(* IEC 61131-3 sources: beckhoffAutomationInterface/ST/Shark/Lib/Controllers/Temperature, 7 files *)

(* ---- GVL_HeatZone.st ---- *)
(* Compile-time bounds for FB_HeatZone arrays.
   MAX_CHANNELS sizes the per-zone channel arrays (the zone's _aipChannels).
   A "channel" is one RTD + one SSR + one PID controller pair.
   Pick the smallest bound that covers the largest physical heat zone on any
   supported machine. PRO DALP currently has 7 channels; 8 leaves headroom. *)
{attribute 'qualified_only'}
VAR_GLOBAL CONSTANT
    MAX_CHANNELS : INT := 8;   // Maximum channels per heat zone
END_VAR

(* ---- FB_BeckhoffTempController.st ---- *)
(* Beckhoff temperature controller for single heating zone. Integrates dual sensor support, PID control, and safety monitoring. *)
FUNCTION_BLOCK FB_BeckhoffTempController IMPLEMENTS I_Tunable
VAR_OUTPUT
    stStatus : ST_BeckhoffTempZoneStatus;  // Consolidated status (all-in-one)
END_VAR
VAR
    // Configuration
    _stConfig : ST_BeckhoffTempZoneConfig;
    _bInitialized : BOOL := FALSE;

    // Hardware
    _ipTemperatureSensor : I_Sensor;     // Temperature sensor (single or dual)
    _ipHeaterOutput     : I_DigitalOutput;

    // Core components - Direct use of Beckhoff controller
    _fbTempController   : FB_CTRL_TempController;

    // Safety system (heater watchdog only - execution monitoring via TwinCAT task watchdog)
    _fbHeaterWatchdog   : FB_HeaterSafetyWatchdog;

    // Independent over-temperature interlock via an optional safety thermocouple.
    // Defence in depth: measured independently of the control RTD. Wired in via
    // InitSafety(); channels without a safety TC leave _bSafetyMonitorActive FALSE
    // and behave exactly as before.
    _fbOverTempMonitor    : FB_OverTemperatureMonitor;
    _bSafetyMonitorActive : BOOL := FALSE;

    // Control state
    _bEnabled           : BOOL := FALSE;
    _rTargetSetpoint    : LREAL := 0.0;
    _eControlMode       : E_CTRL_MODE := E_CTRL_MODE.eCTRL_MODE_IDLE;
    _bHeaterOutput      : BOOL := FALSE;

    // Quick access
    _rCurrentTemperature : LREAL;                        // Current measured temperature (°C)
    _bSensorError       : BOOL;                         // Cached sensor error state

    // Centralized error handling
    _fbError            : FB_ErrorHandler;

    // Execution health
    _bControllerOK      : BOOL;
    _bSafetyTripped     : BOOL;
END_VAR

METHOD PUBLIC Init : BOOL
VAR_INPUT
    ipTemperatureSensor : I_Sensor;  // Temperature sensor
    ipHeaterOutput      : I_DigitalOutput;      // Heater output
    stConfiguration     : ST_BeckhoffTempZoneConfig; // Zone configuration
END_VAR

    _ipTemperatureSensor := ipTemperatureSensor;
    _ipHeaterOutput := ipHeaterOutput;
    _stConfig := stConfiguration;

    // Use zone ID as error source (identifies which zone has the error)
    _fbError.Init(_stConfig.sZoneID);

    // Initialize watchdog with zone-specific name for error traceability
    _fbHeaterWatchdog.Init(
        sInstanceName := CONCAT('WD_', _stConfig.sZoneID),
        tMaxContinuousOn := stConfiguration.tMaxContinuousOn);

    IF _ipTemperatureSensor = 0 OR _ipHeaterOutput = 0 THEN
        RETURN;
    END_IF

    IF NOT _ValidateConfiguration() THEN
        RETURN;
    END_IF

    // Set control mode based on configuration
    IF stConfiguration.stControllerParams.tCtrlCycleTime = T#0S THEN
        _eControlMode := E_CTRL_MODE.eCTRL_MODE_TUNE;
    ELSE
        _eControlMode := E_CTRL_MODE.eCTRL_MODE_ACTIVE;
    END_IF

    IF _stConfig.bAutoEnable AND _eControlMode = E_CTRL_MODE.eCTRL_MODE_ACTIVE THEN
        _bEnabled := TRUE;
    END_IF

    _bInitialized := TRUE;
    Init := TRUE;

END_METHOD

(* Optional: attach an independent safety thermocouple over-temperature interlock.
   Call after Init(). The trip limit and reset hysteresis come from the controller
   configuration (set at Init); only the sensor interface is injected here, keeping
   hardware wiring (param) separate from configuration (struct). Channels with no
   safety TC simply never call this, or call it with rSafetyTcTripLimit <= 0, and
   keep their existing behaviour. The TC sensor lifecycle (Execute) is owned by the
   wiring program; this controller only reads it through the monitor. Fail-safe on
   TC fault is a fixed policy (always trip). *)
METHOD PUBLIC InitSafety : BOOL
VAR_INPUT
    ipSafetyTc : I_Sensor;     // Independent safety thermocouple (hardware injection)
END_VAR
    IF NOT _bInitialized THEN RETURN; END_IF
    IF ipSafetyTc = 0 THEN RETURN; END_IF
    IF _stConfig.rSafetyTcTripLimit <= 0.0 THEN RETURN; END_IF   // not configured for this channel

    IF NOT _fbOverTempMonitor.Init(
        sInstanceName           := CONCAT('OTM_', _stConfig.sZoneID),
        ipSafetyTc              := ipSafetyTc,
        rTripLimit              := _stConfig.rSafetyTcTripLimit,
        rResetHysteresis        := _stConfig.rSafetyTcResetHysteresis,
        bTreatSensorFaultAsTrip := TRUE)   // fixed fail-safe policy: TC fault is always a trip
    THEN
        RETURN;
    END_IF

    _bSafetyMonitorActive := TRUE;
    InitSafety := TRUE;
END_METHOD

METHOD PUBLIC Execute : BOOL
VAR
    eActiveMode : E_CTRL_MODE;
END_VAR

    IF NOT _bInitialized THEN
        IF _ipHeaterOutput <> 0 THEN _ipHeaterOutput.SetOutput(FALSE);
        END_IF
        RETURN;
    END_IF

    // 1. Read Inputs
    _rCurrentTemperature := _ipTemperatureSensor.GetMeasurement();
    _bSensorError := _ipTemperatureSensor.IsError();

    _fbHeaterWatchdog.bHeaterState := _ipHeaterOutput.GetOutput();
    _fbHeaterWatchdog.bManualTrip := FALSE;
    _fbHeaterWatchdog.Execute();

    // Independent over-temperature interlock (optional safety thermocouple)
    IF _bSafetyMonitorActive THEN
        _fbOverTempMonitor.Execute();
    END_IF

    // 2. Determine Safety State (includes over-temperature protection)
    _bSafetyTripped := _fbHeaterWatchdog.IsTripActive()
    OR _bSensorError
    OR (_rCurrentTemperature > _stConfig.rSafetyMaxTemp)
    OR (_bSafetyMonitorActive AND _fbOverTempMonitor.IsTripActive());

    // 3. Determine Control Mode
    IF _eControlMode = E_CTRL_MODE.eCTRL_MODE_RESET THEN
        // Allow RESET command to pass through regardless of enable state
        eActiveMode := E_CTRL_MODE.eCTRL_MODE_RESET;
    ELSIF _bSafetyTripped OR NOT _bEnabled THEN
        eActiveMode := E_CTRL_MODE.eCTRL_MODE_IDLE;
    ELSE
        eActiveMode := _eControlMode;
    END_IF

    // 4. Execute Controller
    _fbTempController(
        eCtrlMode := eActiveMode,
        bSelSetpoint := FALSE,
        fW1 := _rTargetSetpoint,
        fX := _rCurrentTemperature,
        fYManual := _stConfig.rOutputSafeDefault,
        bOpenThermocouple := FALSE,
        bReverseThermocouple := FALSE,
        bBackVoltage := FALSE,
        bLeakage := FALSE,
        bShortCircuit := FALSE,
        bOpenCircuit := FALSE,
        sParaControllerExternal := _stConfig.stExternalPID,
        sControllerParameter := _stConfig.stControllerParams
    );

    _bControllerOK := NOT _fbTempController.bError;

    // 5. Update Outputs (Safety Override)
    _bHeaterOutput := _fbTempController.bYPWMPos AND NOT _bSafetyTripped AND _bControllerOK;

    IF _ipHeaterOutput <> 0 THEN
        _ipHeaterOutput.SetOutput(_bHeaterOutput);
    END_IF

    // 6. Update Status
    _UpdateStatus();

    Execute := NOT _bSafetyTripped;

END_METHOD

METHOD PUBLIC SetSetpoint : BOOL
VAR_INPUT
    rDesiredSetpoint : LREAL;                           // Desired temperature (°C)
END_VAR

    IF rDesiredSetpoint >= _stConfig.rMinSetpoint AND rDesiredSetpoint <= _stConfig.rMaxSetpoint THEN
        _rTargetSetpoint := rDesiredSetpoint;
        SetSetpoint := TRUE;
    END_IF

END_METHOD

METHOD PUBLIC Enable : BOOL
VAR_INPUT
    bEnable : BOOL;
END_VAR

    IF NOT _bSafetyTripped THEN
        _bEnabled := bEnable;

        // Auto-recovery: If enabling, ensure we are in ACTIVE mode if currently in IDLE or RESET
        // IMPORTANT: Do NOT auto-switch if in TUNE mode (would interfere with tuning or coordinator)
        IF bEnable AND (_eControlMode = E_CTRL_MODE.eCTRL_MODE_IDLE OR _eControlMode = E_CTRL_MODE.eCTRL_MODE_RESET) THEN
            _eControlMode := E_CTRL_MODE.eCTRL_MODE_ACTIVE;
        END_IF

        Enable := TRUE;
    ELSE
        _bEnabled := FALSE;
    END_IF

END_METHOD

METHOD PUBLIC Reset : BOOL
VAR
    bWatchdogReset : BOOL;
    bMonitorReset  : BOOL := TRUE;
END_VAR

    bWatchdogReset := _fbHeaterWatchdog.Reset();

    // Cascade the reset to the over-temperature interlock when present
    IF _bSafetyMonitorActive THEN
        bMonitorReset := _fbOverTempMonitor.Reset();
    END_IF

    Reset := bWatchdogReset AND bMonitorReset;

    // Reset controller by setting mode
    SetControlMode(E_CTRL_MODE.eCTRL_MODE_RESET);

    ClearError();

    IF Reset THEN
        _bSafetyTripped := FALSE;
    END_IF

END_METHOD

    // Error Handling Methods

METHOD PRIVATE RaiseError
VAR_INPUT
    eErrorId : E_ErrorId;
    sMessage : STRING(255);
END_VAR
    _fbError.Raise(eErrorId, sMessage);
    stStatus.stError := _fbError.GetError();
END_METHOD

METHOD PRIVATE ClearError
    IF _fbError.IsActive() THEN
        _fbError.Clear();
        stStatus.stError := _fbError.GetError();
    END_IF
END_METHOD

METHOD PRIVATE _UpdateStatus
VAR
    sCtrlErrorMsg : STRING(255);
END_VAR
    // Basic State
    stStatus.bEnabled := _bEnabled;
    stStatus.rSetpoint := _rTargetSetpoint;
    stStatus.rMeasuredValue := _rCurrentTemperature;
    stStatus.rOutput := _fbTempController.fYAnalog;
    stStatus.eCtrlState := _fbTempController.eCtrlState;
    stStatus.bHeaterActive := _fbTempController.bYPWMPos;
    stStatus.rPWMOutput := stStatus.rOutput;
    stStatus.sZoneID := _stConfig.sZoneID;
    stStatus.bSafetyTripped := _bSafetyTripped;
    stStatus.bSensorOK := NOT _bSensorError;
    stStatus.bControllerOK := _bControllerOK;
    // stStatus.bHealthy is updated below

    // Setpoint Reached Check - use common utility function
    stStatus.bAtSetpoint := F_IsWithinAbsoluteTolerance(
        rMeasured := _rCurrentTemperature,
        rSetpoint := _rTargetSetpoint,
        rToleranceAbsolute := _stConfig.rSetpointTolerance,
        bEnabled := _bEnabled AND stStatus.bSensorOK AND NOT _bSafetyTripped
    );

    // Health Check
    stStatus.bHealthy := _bInitialized
    AND stStatus.bSensorOK
    AND _bControllerOK
    AND NOT _bSafetyTripped;

    // Error Detail - Update error based on current conditions
    IF _rCurrentTemperature > _stConfig.rSafetyMaxTemp THEN
        _fbError.RaiseWithValues(E_ErrorId.ERR_CTRL_LIMIT_EXCEEDED, 'Temp', _rCurrentTemperature, _stConfig.rSafetyMaxTemp, 'C');
        stStatus.stError := _fbError.GetError();
        stStatus.bCanResetSafety := (_rCurrentTemperature < _stConfig.rSafetyMaxTemp);
        stStatus.sBlockReason := 'Over-temperature';
    ELSIF _bSafetyMonitorActive AND _fbOverTempMonitor.IsTripActive() THEN
        // Independent safety-thermocouple over-temperature interlock. Inert on
        // machines that never call InitSafety (_bSafetyMonitorActive = FALSE), so
        // this branch only runs where a TC is actually fitted. Surface the
        // monitor's own error so the zone rollup reports the true TC cause.
        _fbError.RaiseFromChild(_fbOverTempMonitor.GetError());
        stStatus.stError := _fbError.GetError();
        stStatus.bCanResetSafety := _fbOverTempMonitor.CanReset();
        stStatus.sBlockReason := _fbOverTempMonitor.GetBlockReason();
    ELSIF _fbHeaterWatchdog.IsTripActive() THEN
        _fbError.RaiseFromChild(_fbHeaterWatchdog.GetError());
        stStatus.stError := _fbError.GetError();
        stStatus.bCanResetSafety := _fbHeaterWatchdog.CanReset();
        stStatus.sBlockReason := _fbHeaterWatchdog.GetBlockReason();
    ELSIF NOT stStatus.bSensorOK THEN
        _fbError.RaiseFromChild(_ipTemperatureSensor.GetError());
        stStatus.stError := _fbError.GetError();
        stStatus.bCanResetSafety := FALSE;
        stStatus.sBlockReason := 'Sensor fault';
    ELSIF _fbTempController.bError THEN
        sCtrlErrorMsg := CONCAT('Controller internal error: ', TO_STRING(_fbTempController.eErrorId));
        RaiseError(E_ErrorId.ERR_GEN_INTERNAL, sCtrlErrorMsg);
        stStatus.bCanResetSafety := FALSE;
        stStatus.sBlockReason := 'Controller error';
    ELSE
        // Clear error when all conditions are OK
        ClearError();
        stStatus.bCanResetSafety := FALSE;
        stStatus.sBlockReason := '';
    END_IF

END_METHOD

METHOD PUBLIC SetControlMode : BOOL
VAR_INPUT
    eMode : E_CTRL_MODE;
END_VAR

    IF NOT _bInitialized THEN RETURN;
    END_IF

    _eControlMode := eMode;
    SetControlMode := TRUE;
END_METHOD

METHOD PUBLIC GetControlMode : E_CTRL_MODE
    GetControlMode := _eControlMode;
END_METHOD

METHOD PUBLIC GetStatus : ST_ControllerStatus
    GetStatus := stStatus;
END_METHOD

METHOD PUBLIC GetZoneStatus : ST_BeckhoffTempZoneStatus
    GetZoneStatus := stStatus;
END_METHOD

    // Ramp Rate Methods

METHOD PUBLIC SetHeatingRampRate : BOOL
VAR_INPUT
    rRate_DegPerMin : LREAL;  // Ramp rate in °C per minute (0 = instant)
END_VAR
    IF NOT _bInitialized THEN RETURN;
    END_IF

    _stConfig.stControllerParams.fWVeloPos := F_RampRateToVelocity(rRate_DegPerMin);
    SetHeatingRampRate := TRUE;
END_METHOD

METHOD PUBLIC SetCoolingRampRate : BOOL
VAR_INPUT
    rRate_DegPerMin : LREAL;  // Ramp rate in °C per minute (0 = instant)
END_VAR
    IF NOT _bInitialized THEN RETURN;
    END_IF

    _stConfig.stControllerParams.fWVeloNeg := F_RampRateToVelocity(rRate_DegPerMin);
    SetCoolingRampRate := TRUE;
END_METHOD

METHOD PUBLIC GetHeatingRampRate : LREAL
    IF _bInitialized THEN
        GetHeatingRampRate := F_VelocityToRampRate(_stConfig.stControllerParams.fWVeloPos);
    ELSE
        GetHeatingRampRate := 0.0;
    END_IF
END_METHOD

METHOD PUBLIC GetCoolingRampRate : LREAL
    IF _bInitialized THEN
        GetCoolingRampRate := F_VelocityToRampRate(_stConfig.stControllerParams.fWVeloNeg);
    ELSE
        GetCoolingRampRate := 0.0;
    END_IF
END_METHOD

METHOD PRIVATE _ValidateConfiguration : BOOL
    IF _stConfig.rMinSetpoint >= _stConfig.rMaxSetpoint THEN
        RaiseError(E_ErrorId.ERR_GEN_INVALID_PARAM, 'Min setpoint must be less than max');
        RETURN;
    END_IF

    IF _stConfig.rSafetyMaxTemp <= _stConfig.rMaxSetpoint THEN
        RaiseError(E_ErrorId.ERR_GEN_INVALID_PARAM, 'Safety max must exceed max setpoint');
        RETURN;
    END_IF

    IF _stConfig.rAbsoluteMaxTemp <= _stConfig.rSafetyMaxTemp THEN
        RaiseError(E_ErrorId.ERR_GEN_INVALID_PARAM, 'Absolute max must exceed safety max');
        RETURN;
    END_IF

    IF _stConfig.rSetpointTolerance <= 0.0 THEN
        RaiseError(E_ErrorId.ERR_GEN_INVALID_PARAM, 'Setpoint tolerance must be positive');
        RETURN;
    END_IF

    _ValidateConfiguration := TRUE;
END_METHOD

END_FUNCTION_BLOCK

(* ---- FB_BeckhoffTuningPanel.st ---- *)
(* Generic PID tuning panel — machine-agnostic.

Operates polymorphically on an I_Tunable, which may be a whole heat zone
(all channels autotuned simultaneously) or a single channel. The owning PRG
resolves the HMI selection (zone idx + channel idx + whole-zone flag) into the
correct I_Tunable via the temperature subsystem and injects it via ipTunable.

Zone vs single-channel tuning is the operator's choice; default is whole-zone
(bTuneWholeZone := TRUE), so every channel in the selected zone tunes at once.

Workflow:
  1. HMI selects iSelectedZoneIdx (+ iSelectedChannelIdx, bTuneWholeZone).
  2. HMI sets rTuningSetpoint.
  3. HMI sets bEnableTuning := TRUE  -> panel latches the current target,
     switches it to TUNE mode, applies the setpoint, and enables it.
  4. Operator monitors stStatus until the autotune converges.
  5. HMI sets bEnableTuning := FALSE -> panel disables the target and
     restores ACTIVE mode.

The target is latched at enable time (_ipActive), so changing the selection
while a tune is running cannot orphan the controller being tuned: the latched
target keeps running until the operator disables tuning. *)
FUNCTION_BLOCK FB_BeckhoffTuningPanel
VAR_INPUT
    ipTunable : I_Tunable;   // Resolved by the owning PRG from the selection fields below
END_VAR
VAR
    // --- HMI selection (read by the owning PRG to resolve ipTunable) ---
    iSelectedZoneIdx    : INT := 1;      // 1..N zone index (maps 1:1 to E_HeatZone)
    iSelectedChannelIdx : INT := 1;      // 1..M channel within the zone (single-channel mode)
    bTuneWholeZone      : BOOL := TRUE;  // TRUE = tune every channel in the zone at once

    // --- HMI commands ---
    rTuningSetpoint     : LREAL := 0.0;  // Target temperature for tuning (°C)
    bEnableTuning       : BOOL;          // Level: TRUE = run autotune on the selection
    bCmdApply           : BOOL;          // One-shot: re-apply the setpoint
    bCmdReset           : BOOL;          // One-shot: reset the target controller

    // --- HMI status ---
    stStatus            : ST_ControllerStatus;  // Live status of the active (or preview) target
    bTuningActive       : BOOL;                 // TRUE while a tune is latched and running
    bReady              : BOOL;                 // TRUE when an I_Tunable is injected
    eActiveMode         : E_CTRL_MODE;          // Current mode of the active (or preview) target

    // --- Internal ---
    _ipActive           : I_Tunable;   // Latched target while tuning (prevents orphaning)
    _bLastEnableTuning  : BOOL;
END_VAR

    bReady := (ipTunable <> 0);

    // ----- Rising edge: latch target and enter TUNE -----
    IF bEnableTuning AND NOT _bLastEnableTuning AND bReady THEN
        _ipActive := ipTunable;
        _ipActive.SetControlMode(E_CTRL_MODE.eCTRL_MODE_TUNE);
        _ipActive.SetSetpoint(rTuningSetpoint);
        _ipActive.Enable(TRUE);
        bTuningActive := TRUE;
    END_IF

    // ----- Falling edge: exit TUNE and restore ACTIVE (keep enabled — use manual panel to disable) -----
    IF (NOT bEnableTuning) AND _bLastEnableTuning AND (_ipActive <> 0) THEN
        _ipActive.SetControlMode(E_CTRL_MODE.eCTRL_MODE_ACTIVE);
        _ipActive := 0;
        bTuningActive := FALSE;
    END_IF

    _bLastEnableTuning := bEnableTuning;

    // ----- One-shot commands: act on the latched target while tuning -----
    IF bTuningActive AND (_ipActive <> 0) THEN
        IF bCmdApply THEN
            _ipActive.SetSetpoint(rTuningSetpoint);
            bCmdApply := FALSE;
        END_IF
        IF bCmdReset THEN
            _ipActive.Reset();
            bCmdReset := FALSE;
        END_IF
    ELSE
        // Not tuning — clear one-shots so they cannot fire on the next enable
        bCmdApply := FALSE;
        bCmdReset := FALSE;
    END_IF

    // ----- Status: latched target while tuning, else live preview of the selection -----
    IF bTuningActive AND (_ipActive <> 0) THEN
        stStatus    := _ipActive.GetStatus();
        eActiveMode := _ipActive.GetControlMode();
    ELSIF bReady THEN
        stStatus    := ipTunable.GetStatus();
        eActiveMode := ipTunable.GetControlMode();
    END_IF

END_FUNCTION_BLOCK

(* ---- FB_HeaterSafetyWatchdog.st ---- *)
(* Heater safety watchdog for runaway heating protection. Monitors continuous heater ON time and manual emergency trip. *)
FUNCTION_BLOCK FB_HeaterSafetyWatchdog
VAR_INPUT
    bHeaterState         : BOOL;                // Current heater output state
    bManualTrip          : BOOL := FALSE;       // Emergency stop button
END_VAR
VAR_OUTPUT
    bTripActive          : BOOL;                // TRUE = force heater OFF
END_VAR
VAR
    _tMaxContinuousOn    : TIME := T#5M;
    _tMinOffTime         : TIME := T#5S;

    _tonContinuousOn     : TON;
    _tonOffTime          : TON;

    _bTripLatched        : BOOL := FALSE;
    _fbError             : FB_ErrorHandler;
    _bCanReset           : BOOL := FALSE;
    _sBlockReason        : STRING(80) := '';
    _bInitialized        : BOOL := FALSE;
END_VAR

METHOD PUBLIC Init : BOOL
VAR_INPUT
    sInstanceName    : STRING(80);
    tMaxContinuousOn : TIME := T#5M;
    tMinOffTime      : TIME := T#5S;
END_VAR
    _fbError.Init(sInstanceName);
    _tMaxContinuousOn := tMaxContinuousOn;
    _tMinOffTime := tMinOffTime;
    _bInitialized := TRUE;
    Init := TRUE;
END_METHOD

METHOD PUBLIC Execute : BOOL
VAR
    rMaxOnSeconds : LREAL;
    rOnSeconds    : LREAL;
END_VAR
    IF NOT _bInitialized THEN
        RETURN;
    END_IF

    // 1. Monitor CONTINUOUS ON time (resets when heater cycles OFF)
    _tonContinuousOn(IN := bHeaterState AND NOT _bTripLatched, PT := _tMaxContinuousOn);

    // Trip if heater stuck ON continuously
    IF _tonContinuousOn.Q AND NOT _bTripLatched THEN
        _bTripLatched := TRUE;
        rMaxOnSeconds := TIME_TO_LREAL(_tMaxContinuousOn) / 1000.0;
        rOnSeconds := TIME_TO_LREAL(_tonContinuousOn.ET) / 1000.0;
        _fbError.RaiseWithValues(E_ErrorId.ERR_CTRL_WATCHDOG_HEATING, 'OnTime', rOnSeconds, rMaxOnSeconds, 's');
    END_IF

    // 2. Manual emergency trip
    IF bManualTrip AND NOT _bTripLatched THEN
        _bTripLatched := TRUE;
        _fbError.Raise(E_ErrorId.ERR_CTRL_LIMIT_EXCEEDED, 'Manual emergency trip activated');
    END_IF

    // 3. Track time since trip (for minimum OFF time enforcement)
    _tonOffTime(IN := _bTripLatched, PT := _tMinOffTime);

    // 4. Determine if reset is allowed
    _bCanReset := NOT bHeaterState           // Heater must be OFF
    AND _tonOffTime.Q              // Minimum OFF time elapsed
    AND _bTripLatched;             // Only when tripped

    // 5. Update block reason
    IF NOT _bTripLatched THEN
        _sBlockReason := '';
    ELSIF bHeaterState THEN
        _sBlockReason := 'Heater still ON';
    ELSIF NOT _tonOffTime.Q THEN
        _sBlockReason := 'Minimum OFF time not elapsed';
    ELSE
        _sBlockReason := '';
    END_IF

    // 6. Update outputs
    bTripActive := _bTripLatched;
    Execute := NOT bTripActive;

END_METHOD

METHOD PUBLIC Reset : BOOL
    IF NOT _bTripLatched THEN
        Reset := TRUE;  // Already clear
        RETURN;
    END_IF

    IF _bCanReset THEN
        _bTripLatched := FALSE;
        _fbError.Clear();
        _tonContinuousOn(IN := FALSE);  // Reset timer
        _sBlockReason := '';
        Reset := TRUE;
    ELSE
        Reset := FALSE;
    END_IF
END_METHOD

METHOD PUBLIC GetError : ST_Error
    GetError := _fbError.GetError();
END_METHOD

METHOD PUBLIC CanReset : BOOL
    CanReset := _bCanReset;
END_METHOD

METHOD PUBLIC GetBlockReason : STRING(80)
    GetBlockReason := _sBlockReason;
END_METHOD

METHOD PUBLIC IsTripActive : BOOL
    IsTripActive := bTripActive;
END_METHOD

END_FUNCTION_BLOCK

(* ---- FB_HeatJacket.st ---- *)
(*
FB_HeatZone — composite heat zone made of N independent channel controllers.

Each channel owns its own RTD + SSR + PID (e.g. an FB_BeckhoffTempController).
The zone itself does NOT close a control loop. It coordinates:
  * one setpoint pushed to all channels
  * aggregated readback (avg/max/min/master) for the HMI
  * delta safety (auto-disable if channels drift apart)
  * rolled-up health (any channel fault → zone fault)

Implements I_Controller, so a zone and a single channel controller are
interchangeable from the subsystem's point of view. A 1-channel zone
is a valid, minimal-overhead wrapper around one channel.
*)
FUNCTION_BLOCK FB_HeatZone IMPLEMENTS I_Controller
VAR_OUTPUT
    stStatus : ST_HeatZoneStatus;     // Rich aggregated status (zone-specific)
END_VAR
VAR
    _stConfig      : ST_HeatZoneConfig;
    _aipChannels   : ARRAY[1..GVL_HeatZone.MAX_CHANNELS] OF I_Controller;
    _nChannelCount : INT;

    _bInitialized  : BOOL := FALSE;
    _bEnabledCmd   : BOOL := FALSE;     // Last commanded Enable() (before delta-trip override)
    _rSetpointCmd  : LREAL := 0.0;      // Last commanded SetSetpoint()
    _bDeltaTripped : BOOL := FALSE;     // Latched; cleared by Reset()

    _fbError       : FB_ErrorHandler;

    // Cached I_Controller status (rebuilt every Execute)
    _stCtrlStatus  : ST_ControllerStatus;
END_VAR

// ============================================================================
// PUBLIC API
// ============================================================================

METHOD PUBLIC Init : BOOL
VAR_INPUT
    stConfig      : ST_HeatZoneConfig;
    aipChannels   : ARRAY[1..GVL_HeatZone.MAX_CHANNELS] OF I_Controller;
    nChannelCount : INT;
END_VAR
VAR
    i : INT;
END_VAR

    _fbError.Init(stConfig.sZoneID);

    // Validate channel count
    IF nChannelCount < 1 OR nChannelCount > GVL_HeatZone.MAX_CHANNELS THEN
        _fbError.Raise(E_ErrorId.ERR_GEN_INVALID_PARAM, 'Zone channel count out of range');
        RETURN;
    END_IF

    // Validate every channel pointer is non-null
    FOR i := 1 TO nChannelCount DO
        IF aipChannels[i] = 0 THEN
            _fbError.Raise(E_ErrorId.ERR_GEN_NULL_POINTER, 'Zone channel pointer is null');
            RETURN;
        END_IF
    END_FOR

    // Validate setpoint clamp
    IF stConfig.rMinSetpoint >= stConfig.rMaxSetpoint THEN
        _fbError.Raise(E_ErrorId.ERR_GEN_INVALID_PARAM, 'Zone min setpoint must be less than max');
        RETURN;
    END_IF

    // Copy in
    _stConfig := stConfig;
    _nChannelCount := nChannelCount;
    FOR i := 1 TO nChannelCount DO
        _aipChannels[i] := aipChannels[i];
    END_FOR

    stStatus.sZoneID := stConfig.sZoneID;
    stStatus.nChannelCount := nChannelCount;

    _bInitialized := TRUE;
    Init := TRUE;
END_METHOD

METHOD PUBLIC Execute : BOOL
    IF NOT _bInitialized THEN RETURN; END_IF

    _ReadChannels();
    _ApplyDeltaTrip();
    _UpdateCtrlStatus();

    Execute := NOT stStatus.bAnyError AND NOT _bDeltaTripped;
END_METHOD

{attribute 'estimated-stack-usage' := '500'}
METHOD PUBLIC Enable : BOOL
VAR_INPUT
    bEnable : BOOL;
END_VAR
VAR
    i : INT;
    ipChannel : I_Controller;
END_VAR
    IF NOT _bInitialized THEN RETURN; END_IF

    // Refuse to enable while delta-tripped; disable always allowed
    IF bEnable AND _bDeltaTripped THEN
        Enable := FALSE;
        RETURN;
    END_IF

    _bEnabledCmd := bEnable;

    FOR i := 1 TO _nChannelCount DO
        ipChannel := _aipChannels[i];
        ipChannel.Enable(bEnable);
    END_FOR

    Enable := TRUE;
END_METHOD

{attribute 'estimated-stack-usage' := '500'}
METHOD PUBLIC SetSetpoint : BOOL
VAR_INPUT
    rDesiredSetpoint : LREAL;
END_VAR
VAR
    i : INT;
    ipChannel : I_Controller;
END_VAR
    IF NOT _bInitialized THEN RETURN; END_IF

    // Zone-level clamp; channel-level clamp still applies inside each channel
    IF rDesiredSetpoint < _stConfig.rMinSetpoint OR rDesiredSetpoint > _stConfig.rMaxSetpoint THEN
        SetSetpoint := FALSE;
        RETURN;
    END_IF

    _rSetpointCmd := rDesiredSetpoint;

    FOR i := 1 TO _nChannelCount DO
        ipChannel := _aipChannels[i];
        ipChannel.SetSetpoint(rDesiredSetpoint);
    END_FOR

    SetSetpoint := TRUE;
END_METHOD

{attribute 'estimated-stack-usage' := '500'}
METHOD PUBLIC Reset : BOOL
VAR
    i : INT;
    bAllOk : BOOL := TRUE;
    ipChannel : I_Controller;
END_VAR
    IF NOT _bInitialized THEN RETURN; END_IF

    FOR i := 1 TO _nChannelCount DO
        ipChannel := _aipChannels[i];
        IF NOT ipChannel.Reset() THEN
            bAllOk := FALSE;
        END_IF
    END_FOR

    _bDeltaTripped := FALSE;
    stStatus.bDeltaTripped := FALSE;
    _fbError.Clear();

    Reset := bAllOk;
END_METHOD

METHOD PUBLIC GetStatus : ST_ControllerStatus
    GetStatus := _stCtrlStatus;
END_METHOD

// ----------------------------------------------------------------------------
// Diagnostics accessors (zone-specific; outside I_Controller surface)
// ----------------------------------------------------------------------------

METHOD PUBLIC GetChannel : I_Controller
VAR_INPUT
    nIndex : INT;   // 1..nChannelCount
END_VAR
    IF nIndex >= 1 AND nIndex <= _nChannelCount THEN
        GetChannel := _aipChannels[nIndex];
    ELSE
        GetChannel := 0;
    END_IF
END_METHOD

METHOD PUBLIC GetChannelCount : INT
    GetChannelCount := _nChannelCount;
END_METHOD

// ============================================================================
// PRIVATE
// ============================================================================

METHOD PRIVATE _ReadChannels
VAR
    i              : INT;
    stCh           : ST_ControllerStatus;
    rSum           : LREAL := 0.0;
    rTemp          : LREAL;
    bAllAt         : BOOL := TRUE;
    bAnyErr        : BOOL := FALSE;
    nFirstErr      : INT := 0;
    stFirstErr     : ST_Error;
END_VAR
    // Seed min/max with the first channel so SEL works for all N (incl. N=1)
    stCh := _aipChannels[1].GetStatus();
    stStatus.rMin := stCh.rMeasuredValue;
    stStatus.rMax := stCh.rMeasuredValue;
    stStatus.nColdestIdx := 1;
    stStatus.nHottestIdx := 1;

    FOR i := 1 TO _nChannelCount DO
        stCh := _aipChannels[i].GetStatus();
        rTemp := stCh.rMeasuredValue;
        rSum := rSum + rTemp;

        IF rTemp < stStatus.rMin THEN
            stStatus.rMin := rTemp;
            stStatus.nColdestIdx := i;
        END_IF
        IF rTemp > stStatus.rMax THEN
            stStatus.rMax := rTemp;
            stStatus.nHottestIdx := i;
        END_IF

        IF NOT stCh.bAtSetpoint THEN
            bAllAt := FALSE;
        END_IF

        IF stCh.stError.eErrorId <> E_ErrorId.NO_ERROR THEN
            IF NOT bAnyErr THEN
                nFirstErr := i;
                stFirstErr := stCh.stError;
            END_IF
            bAnyErr := TRUE;
        END_IF
    END_FOR

    // Aggregation
    CASE _stConfig.eAggregation OF
        E_TempAggregation.AVERAGE:
            stStatus.rAggregated := rSum / TO_LREAL(_nChannelCount);
        E_TempAggregation.MAXIMUM:
            stStatus.rAggregated := stStatus.rMax;
        E_TempAggregation.MINIMUM:
            stStatus.rAggregated := stStatus.rMin;
        E_TempAggregation.MASTER:
            stCh := _aipChannels[1].GetStatus();
            stStatus.rAggregated := stCh.rMeasuredValue;
    ELSE
        stStatus.rAggregated := rSum / TO_LREAL(_nChannelCount);
    END_CASE

    stStatus.rDelta := stStatus.rMax - stStatus.rMin;
    stStatus.rSetpoint := _rSetpointCmd;
    stStatus.bAllAtSetpoint := bAllAt AND _bEnabledCmd;
    stStatus.bAnyError := bAnyErr;
    stStatus.nFirstErrorIdx := nFirstErr;
    stStatus.stFirstError := stFirstErr;
    stStatus.bDeltaWarning := (_stConfig.rMaxDeltaWarn > 0.0)
                             AND (stStatus.rDelta > _stConfig.rMaxDeltaWarn);
END_METHOD

METHOD PRIVATE _ApplyDeltaTrip
VAR
    i : INT;
END_VAR
    // Already tripped — stays latched until Reset()
    IF _bDeltaTripped THEN RETURN; END_IF

    // Trip disabled (rMaxDeltaTrip = 0) or zone not enabled — skip
    IF _stConfig.rMaxDeltaTrip <= 0.0 OR NOT _bEnabledCmd THEN RETURN; END_IF

    IF stStatus.rDelta > _stConfig.rMaxDeltaTrip THEN
        _bDeltaTripped := TRUE;
        stStatus.bDeltaTripped := TRUE;
        _fbError.RaiseWithValues(
            E_ErrorId.ERR_CTRL_LIMIT_EXCEEDED,
            'ZoneDelta',
            stStatus.rDelta,
            _stConfig.rMaxDeltaTrip,
            'C');

        // Disable every channel (override commanded enable)
        FOR i := 1 TO _nChannelCount DO
            _aipChannels[i].Enable(FALSE);
        END_FOR
    END_IF
END_METHOD

METHOD PRIVATE _UpdateCtrlStatus
    // Build the polymorphic ST_ControllerStatus surface for I_Controller callers
    _stCtrlStatus.rMeasuredValue := stStatus.rAggregated;
    _stCtrlStatus.rSetpoint      := stStatus.rSetpoint;
    _stCtrlStatus.rOutput        := 0.0;   // Per-channel; not meaningful at zone level
    _stCtrlStatus.bEnabled       := _bEnabledCmd AND NOT _bDeltaTripped;
    _stCtrlStatus.bAtSetpoint    := stStatus.bAllAtSetpoint;

    IF _bDeltaTripped THEN
        _stCtrlStatus.stError := _fbError.GetError();
    ELSIF stStatus.bAnyError THEN
        _stCtrlStatus.stError := stStatus.stFirstError;
    ELSE
        _stCtrlStatus.stError.eErrorId := E_ErrorId.NO_ERROR;
    END_IF
END_METHOD

END_FUNCTION_BLOCK

(* ---- FB_HeatZone.st ---- *)
(*
FB_HeatZone — composite heat zone made of N independent channel controllers.

Each channel owns its own RTD + SSR + PID (e.g. an FB_BeckhoffTempController).
The zone itself does NOT close a control loop. It coordinates:
  * one setpoint pushed to all channels
  * aggregated readback (avg/max/min/master) for the HMI
  * delta safety (auto-disable if channels drift apart)
  * rolled-up health (any channel fault → zone fault)

Implements I_Controller, so a zone and a single channel controller are
interchangeable from the subsystem's point of view. A 1-channel zone
is a valid, minimal-overhead wrapper around one channel.
*)
FUNCTION_BLOCK FB_HeatZone IMPLEMENTS I_Tunable
VAR_OUTPUT
    stStatus : ST_HeatZoneStatus;     // Rich aggregated status (zone-specific)
END_VAR
VAR
    _stConfig      : ST_HeatZoneConfig;
    _aipChannels   : ARRAY[1..GVL_HeatZone.MAX_CHANNELS] OF I_Tunable;
    _nChannelCount : INT;

    _bInitialized  : BOOL := FALSE;
    _bEnabledCmd   : BOOL := FALSE;     // Last commanded Enable() (before delta-trip override)
    _rSetpointCmd  : LREAL := 0.0;      // Last commanded SetSetpoint()
    _bDeltaTripped : BOOL := FALSE;     // Latched; cleared by Reset()
    _bChannelSafetyTripped : BOOL := FALSE;  // Latched zone trip from a channel safety latch (any cause); cleared by Reset()
    _bAnyChSafetyTrip      : BOOL := FALSE;  // Instantaneous: any channel reported a safety trip this scan
    _nFirstChSafetyTripIdx : INT := 0;       // Instantaneous: first channel with a safety trip this scan
    _stFirstChSafetyError  : ST_Error;       // Actual fault of the first safety-tripped channel (propagated to the zone)
    _bPowerAvailable : BOOL := TRUE;    // External main-power interlock (e.g. MCR). FALSE = power cut:
                                        // force all channels disabled and refuse Enable(TRUE).
    _eZoneMode     : E_CTRL_MODE := E_CTRL_MODE.eCTRL_MODE_ACTIVE;  // Last mode cascaded to channels

    _fbError       : FB_ErrorHandler;

    // Cached I_Controller status (rebuilt every Execute)
    _stCtrlStatus  : ST_ControllerStatus;
END_VAR

// ============================================================================
// PUBLIC API
// ============================================================================

METHOD PUBLIC Init : BOOL
VAR_INPUT
    stConfig      : ST_HeatZoneConfig;
    aipChannels   : ARRAY[1..GVL_HeatZone.MAX_CHANNELS] OF I_Tunable;
    nChannelCount : INT;
END_VAR
VAR
    i : INT;
END_VAR

    _fbError.Init(stConfig.sZoneID);

    // Validate channel count
    IF nChannelCount < 1 OR nChannelCount > GVL_HeatZone.MAX_CHANNELS THEN
        _fbError.Raise(E_ErrorId.ERR_GEN_INVALID_PARAM, 'Zone channel count out of range');
        RETURN;
    END_IF

    // Validate every channel pointer is non-null
    FOR i := 1 TO nChannelCount DO
        IF aipChannels[i] = 0 THEN
            _fbError.Raise(E_ErrorId.ERR_GEN_NULL_POINTER, 'Zone channel pointer is null');
            RETURN;
        END_IF
    END_FOR

    // Validate setpoint clamp
    IF stConfig.rMinSetpoint >= stConfig.rMaxSetpoint THEN
        _fbError.Raise(E_ErrorId.ERR_GEN_INVALID_PARAM, 'Zone min setpoint must be less than max');
        RETURN;
    END_IF

    // Copy in
    _stConfig := stConfig;
    _nChannelCount := nChannelCount;
    FOR i := 1 TO nChannelCount DO
        _aipChannels[i] := aipChannels[i];
    END_FOR

    stStatus.sZoneID := stConfig.sZoneID;
    stStatus.nChannelCount := nChannelCount;

    _bInitialized := TRUE;
    Init := TRUE;
END_METHOD

METHOD PUBLIC Execute : BOOL
    IF NOT _bInitialized THEN RETURN; END_IF

    _ReadChannels();
    _ApplyDeltaTrip();
    _ApplyChannelSafetyTrip();
    _ApplyExternalPowerCut();
    _UpdateCtrlStatus();

    Execute := NOT stStatus.bAnyError AND NOT _bDeltaTripped AND NOT _bChannelSafetyTripped
               AND _bPowerAvailable;
END_METHOD

{attribute 'estimated-stack-usage' := '500'}
METHOD PUBLIC Enable : BOOL
VAR_INPUT
    bEnable : BOOL;
END_VAR
VAR
    i : INT;
    ipChannel : I_Controller;
END_VAR
    IF NOT _bInitialized THEN RETURN; END_IF

    // Refuse to enable while delta-tripped; disable always allowed
    IF bEnable AND _bDeltaTripped THEN
        Enable := FALSE;
        RETURN;
    END_IF

    // Refuse to enable while external main power is cut (e.g. MCR trip);
    // disable is always allowed.
    IF bEnable AND NOT _bPowerAvailable THEN
        Enable := FALSE;
        RETURN;
    END_IF

    _bEnabledCmd := bEnable;

    FOR i := 1 TO _nChannelCount DO
        ipChannel := _aipChannels[i];
        ipChannel.Enable(bEnable);
    END_FOR

    Enable := TRUE;
END_METHOD

{attribute 'estimated-stack-usage' := '500'}
METHOD PUBLIC SetSetpoint : BOOL
VAR_INPUT
    rDesiredSetpoint : LREAL;
END_VAR
VAR
    i : INT;
    ipChannel : I_Controller;
END_VAR
    IF NOT _bInitialized THEN RETURN; END_IF

    // Zone-level clamp; channel-level clamp still applies inside each channel
    IF rDesiredSetpoint < _stConfig.rMinSetpoint OR rDesiredSetpoint > _stConfig.rMaxSetpoint THEN
        SetSetpoint := FALSE;
        RETURN;
    END_IF

    _rSetpointCmd := rDesiredSetpoint;

    FOR i := 1 TO _nChannelCount DO
        ipChannel := _aipChannels[i];
        ipChannel.SetSetpoint(rDesiredSetpoint);
    END_FOR

    SetSetpoint := TRUE;
END_METHOD

{attribute 'estimated-stack-usage' := '500'}
METHOD PUBLIC Reset : BOOL
VAR
    i : INT;
    bAllOk : BOOL := TRUE;
    ipChannel : I_Controller;
END_VAR
    IF NOT _bInitialized THEN RETURN; END_IF

    FOR i := 1 TO _nChannelCount DO
        ipChannel := _aipChannels[i];
        IF NOT ipChannel.Reset() THEN
            bAllOk := FALSE;
        END_IF
    END_FOR

    _bDeltaTripped := FALSE;
    stStatus.bDeltaTripped := FALSE;

    // Clear the channel-safety latch ONLY when every channel actually reset
    // (i.e. each safety TC has cooled below its reset threshold). Clearing it
    // unconditionally would drop bSafetyTripped to FALSE for one cycle before
    // _ApplyChannelSafetyTrip re-latches it — unsafe for a flag external logic
    // may sample. While still tripped we also keep the active error so the HMI
    // continues to show the cause.
    IF bAllOk THEN
        _bChannelSafetyTripped := FALSE;
        stStatus.bSafetyTripped := FALSE;
        stStatus.nSafetyTrippedIdx := 0;
        _fbError.Clear();
    END_IF

    Reset := bAllOk;
END_METHOD

(* External main-power interlock (e.g. an MCR that physically cuts heater mains).
   When bAvailable = FALSE the zone forces every channel disabled each Execute and
   refuses Enable(TRUE), so de-powered channels stop accumulating windup / "heating
   but temperature dropping" errors. This is a live gate, NOT a latch: when power
   returns the zone stays disabled until an operator explicitly re-enables. *)
METHOD PUBLIC SetPowerAvailable : BOOL
VAR_INPUT
    bAvailable : BOOL;
END_VAR
    IF NOT _bInitialized THEN RETURN; END_IF
    _bPowerAvailable := bAvailable;
    SetPowerAvailable := TRUE;
END_METHOD

METHOD PUBLIC GetStatus : ST_ControllerStatus
    GetStatus := _stCtrlStatus;
END_METHOD

// ----------------------------------------------------------------------------
// I_Tunable — cascade the control mode to every channel so an entire zone can
// be put into autotune (or back to ACTIVE) with a single call.
// ----------------------------------------------------------------------------

// FB_HeatZone implements I_Tunable and forwards SetControlMode to its channels,
// which are themselves I_Tunable. The compiler cannot prove a channel is never a
// nested zone, so it treats zone -> I_Tunable.SetControlMode -> zone as potential
// recursion and cannot complete stack analysis (C0298). The recursion is bounded
// by zone-nesting depth (a zone owns leaf channels, so depth is normally 1);
// declare a safe per-call stack estimate so the stack calculation completes.
{attribute 'estimated-stack-usage' := '1000'}
METHOD PUBLIC SetControlMode : BOOL
VAR_INPUT
    eMode : E_CTRL_MODE;
END_VAR
VAR
    i : INT;
END_VAR
    IF NOT _bInitialized THEN RETURN; END_IF

    _eZoneMode := eMode;
    FOR i := 1 TO _nChannelCount DO
        _aipChannels[i].SetControlMode(eMode);
    END_FOR

    SetControlMode := TRUE;
END_METHOD

METHOD PUBLIC GetControlMode : E_CTRL_MODE
    GetControlMode := _eZoneMode;
END_METHOD

// ----------------------------------------------------------------------------
// Diagnostics accessors (zone-specific; outside I_Controller surface)
// ----------------------------------------------------------------------------

METHOD PUBLIC GetChannel : I_Controller
VAR_INPUT
    nIndex : INT;   // 1..nChannelCount
END_VAR
    IF nIndex >= 1 AND nIndex <= _nChannelCount THEN
        GetChannel := _aipChannels[nIndex];
    ELSE
        GetChannel := 0;
    END_IF
END_METHOD

METHOD PUBLIC GetChannelCount : INT
    GetChannelCount := _nChannelCount;
END_METHOD

// ============================================================================
// PRIVATE
// ============================================================================

METHOD PRIVATE _ReadChannels
VAR
    i              : INT;
    stCh           : ST_ControllerStatus;
    rSum           : LREAL := 0.0;
    rTemp          : LREAL;
    bAllAt         : BOOL := TRUE;
    bAnyErr        : BOOL := FALSE;
    nFirstErr      : INT := 0;
    stFirstErr     : ST_Error;
    bAnySafetyTrip : BOOL := FALSE;
    nFirstSafetyTrip : INT := 0;
    stFirstSafetyErr : ST_Error;
END_VAR
    // Seed min/max with the first channel so SEL works for all N (incl. N=1)
    stCh := _aipChannels[1].GetStatus();
    stStatus.rMin := stCh.rMeasuredValue;
    stStatus.rMax := stCh.rMeasuredValue;
    stStatus.nColdestIdx := 1;
    stStatus.nHottestIdx := 1;

    FOR i := 1 TO _nChannelCount DO
        stCh := _aipChannels[i].GetStatus();
        rTemp := stCh.rMeasuredValue;
        rSum := rSum + rTemp;

        IF rTemp < stStatus.rMin THEN
            stStatus.rMin := rTemp;
            stStatus.nColdestIdx := i;
        END_IF
        IF rTemp > stStatus.rMax THEN
            stStatus.rMax := rTemp;
            stStatus.nHottestIdx := i;
        END_IF

        IF NOT stCh.bAtSetpoint THEN
            bAllAt := FALSE;
        END_IF

        IF stCh.stError.eErrorId <> E_ErrorId.NO_ERROR THEN
            IF NOT bAnyErr THEN
                nFirstErr := i;
                stFirstErr := stCh.stError;
            END_IF
            bAnyErr := TRUE;
        END_IF

        IF stCh.bSafetyTripped THEN
            IF NOT bAnySafetyTrip THEN
                nFirstSafetyTrip := i;
                stFirstSafetyErr := stCh.stError;
            END_IF
            bAnySafetyTrip := TRUE;
        END_IF
    END_FOR

    // Aggregation
    CASE _stConfig.eAggregation OF
        E_TempAggregation.AVERAGE:
            stStatus.rAggregated := rSum / TO_LREAL(_nChannelCount);
        E_TempAggregation.MAXIMUM:
            stStatus.rAggregated := stStatus.rMax;
        E_TempAggregation.MINIMUM:
            stStatus.rAggregated := stStatus.rMin;
        E_TempAggregation.MASTER:
            stCh := _aipChannels[1].GetStatus();
            stStatus.rAggregated := stCh.rMeasuredValue;
    ELSE
        stStatus.rAggregated := rSum / TO_LREAL(_nChannelCount);
    END_CASE

    stStatus.rDelta := stStatus.rMax - stStatus.rMin;
    stStatus.rSetpoint := _rSetpointCmd;
    stStatus.bAllAtSetpoint := bAllAt AND _bEnabledCmd;
    stStatus.bAnyError := bAnyErr;
    stStatus.nFirstErrorIdx := nFirstErr;
    stStatus.stFirstError := stFirstErr;
    stStatus.bDeltaWarning := (_stConfig.rMaxDeltaWarn > 0.0)
                             AND (stStatus.rDelta > _stConfig.rMaxDeltaWarn);

    // Hand the instantaneous channel safety detection to _ApplyChannelSafetyTrip
    _bAnyChSafetyTrip      := bAnySafetyTrip;
    _nFirstChSafetyTripIdx := nFirstSafetyTrip;
    _stFirstChSafetyError  := stFirstSafetyErr;
END_METHOD

METHOD PRIVATE _ApplyDeltaTrip
VAR
    i : INT;
END_VAR
    // Skip delta-trip during autotune: each channel runs its own independent PID
    // self-tuning and they intentionally diverge. Per-channel over-temp / watchdog
    // safety stays active inside each FB_BeckhoffTempController.
    IF _eZoneMode = E_CTRL_MODE.eCTRL_MODE_TUNE THEN RETURN; END_IF

    // Already tripped — stays latched until Reset()
    IF _bDeltaTripped THEN RETURN; END_IF

    // Trip disabled (rMaxDeltaTrip = 0) or zone not enabled — skip
    IF _stConfig.rMaxDeltaTrip <= 0.0 OR NOT _bEnabledCmd THEN RETURN; END_IF

    IF stStatus.rDelta > _stConfig.rMaxDeltaTrip THEN
        _bDeltaTripped := TRUE;
        stStatus.bDeltaTripped := TRUE;
        _fbError.RaiseWithValues(
            E_ErrorId.ERR_CTRL_LIMIT_EXCEEDED,
            'ZoneDelta',
            stStatus.rDelta,
            _stConfig.rMaxDeltaTrip,
            'C');

        // Disable every channel (override commanded enable)
        FOR i := 1 TO _nChannelCount DO
            _aipChannels[i].Enable(FALSE);
        END_FOR
    END_IF
END_METHOD

(* Propagate a per-channel safety latch to the whole zone. A channel latches its
   safety state for ANY of: heater watchdog, sensor fault/deviation, control-RTD
   over-temperature, or — where fitted — an independent safety-thermocouple
   over-temperature. Unlike _ApplyDeltaTrip this is NOT suspended during autotune:
   a genuine safety latch is always unsafe, whereas channel divergence is expected
   only for the delta check. The offending channel has already cut its own heater
   (authoritative); this latches the zone so every sibling channel is disabled too
   and an operator Reset() is required. The zone reports the offending channel's
   ACTUAL fault, never a fabricated cause. *)
METHOD PRIVATE _ApplyChannelSafetyTrip
VAR
    i : INT;
END_VAR
    // Feature disabled for this zone — leave channel-local cutoff to act alone
    IF NOT _stConfig.bChannelTripStopsZone THEN RETURN; END_IF

    // Already latched — stays tripped until Reset()
    IF _bChannelSafetyTripped THEN RETURN; END_IF

    // No channel safety trip detected this scan
    IF NOT _bAnyChSafetyTrip THEN RETURN; END_IF

    _bChannelSafetyTripped := TRUE;
    stStatus.bSafetyTripped := TRUE;
    stStatus.nSafetyTrippedIdx := _nFirstChSafetyTripIdx;

    // Propagate the offending channel's ACTUAL fault (sensor deviation, RTD
    // over-temp, heater watchdog, or — where fitted — a safety-TC over-temp)
    // instead of fabricating a fixed "TC over-temperature" reason. The child
    // already logged the root cause; RaiseFromChild carries it up without
    // re-logging, so the zone reports the true reason it disabled.
    _fbError.RaiseFromChild(_stFirstChSafetyError);

    // Disable every channel (override commanded enable)
    FOR i := 1 TO _nChannelCount DO
        _aipChannels[i].Enable(FALSE);
    END_FOR
END_METHOD

(* Force every channel disabled while external main power is cut (e.g. MCR trip).
   Runs every scan (live gate, no latch): the external TwinSAFE project owns the
   trip/reset; we only mirror it so de-powered channels stop trying to heat and
   stop accumulating windup / watchdog errors. Commanded enable is preserved
   internally only insofar as Enable(TRUE) is refused while power is unavailable. *)
METHOD PRIVATE _ApplyExternalPowerCut
VAR
    i : INT;
END_VAR
    IF _bPowerAvailable THEN RETURN; END_IF

    _bEnabledCmd := FALSE;
    FOR i := 1 TO _nChannelCount DO
        _aipChannels[i].Enable(FALSE);
    END_FOR
END_METHOD

METHOD PRIVATE _UpdateCtrlStatus
    // Build the polymorphic ST_ControllerStatus surface for I_Controller callers
    _stCtrlStatus.rMeasuredValue := stStatus.rAggregated;
    _stCtrlStatus.rSetpoint      := stStatus.rSetpoint;
    _stCtrlStatus.rOutput        := 0.0;   // Per-channel; not meaningful at zone level
    _stCtrlStatus.bEnabled       := _bEnabledCmd AND NOT _bDeltaTripped AND NOT _bChannelSafetyTripped
                                    AND _bPowerAvailable;
    _stCtrlStatus.bAtSetpoint    := stStatus.bAllAtSetpoint;
    _stCtrlStatus.bSafetyTripped := _bChannelSafetyTripped;
    stStatus.bExternalPowerCut   := NOT _bPowerAvailable;

    IF _bChannelSafetyTripped OR _bDeltaTripped THEN
        _stCtrlStatus.stError := _fbError.GetError();
    ELSIF stStatus.bAnyError THEN
        _stCtrlStatus.stError := stStatus.stFirstError;
    ELSE
        _stCtrlStatus.stError.eErrorId := E_ErrorId.NO_ERROR;
    END_IF
END_METHOD

END_FUNCTION_BLOCK

(* ---- FB_OverTemperatureMonitor.st ---- *)
(*
FB_OverTemperatureMonitor — independent over-temperature interlock.

Wraps a safety thermocouple (I_Sensor) that is measured independently of the
control RTD, providing defence-in-depth over-temperature protection for one
heat channel. The sensor lifecycle (Execute) is owned by the wiring program;
this monitor only reads it.

Behaviour (mirrors FB_HeaterSafetyWatchdog latch/reset semantics):
  * Trip LATCHES when the TC exceeds rTripLimit.
  * A TC sensor fault is treated as a trip (fail-safe) when
    bTreatSensorFaultAsTrip is TRUE.
  * The trip raises ERR_CTRL_LIMIT_EXCEEDED (logged once via FB_ErrorHandler).
  * Reset() is gated: only allowed once the TC has fallen below
    (rTripLimit - rResetHysteresis) and is fault-free.

The monitor never drives hardware directly — the owning controller reads
IsTripActive() and forces its heater OFF. This keeps the monitor a pure,
side-effect-free safety observer (SRP).
 *)
FUNCTION_BLOCK FB_OverTemperatureMonitor
VAR
    _ipSafetyTc: I_Sensor;
    _rTripLimit: LREAL := 0.0;
    _rResetHysteresis: LREAL := 5.0;
    _bTreatSensorFaultAsTrip: BOOL := TRUE;

    _bTripLatched: BOOL := FALSE;
    _rTemperature: LREAL := 0.0;
    _bSensorFault: BOOL := FALSE;
    _bCanReset: BOOL := FALSE;
    _sBlockReason: STRING(80) := '';
    _fbError: FB_ErrorHandler;
    _bInitialized: BOOL := FALSE;
END_VAR

METHOD PUBLIC Init: BOOL
VAR_INPUT
    sInstanceName: STRING(80);
    ipSafetyTc: I_Sensor; // Independent safety thermocouple
    rTripLimit: LREAL; // Over-temperature trip threshold (°C)
    rResetHysteresis: LREAL := 5.0; // Must cool this far below limit to reset (°C)
    bTreatSensorFaultAsTrip: BOOL := TRUE; // Fail-safe on TC fault
END_VAR
    _fbError.Init(sInstanceName);

    IF ipSafetyTc = 0 THEN
        _fbError.Raise(E_ErrorId.ERR_GEN_NULL_POINTER, 'Safety TC sensor reference is null');
        RETURN;
    END_IF

    IF rTripLimit <= 0.0 THEN
        _fbError.Raise(E_ErrorId.ERR_GEN_INVALID_PARAM, 'Trip limit must be positive');
        RETURN;
    END_IF

    _ipSafetyTc := ipSafetyTc;
    _rTripLimit := rTripLimit;
    _rResetHysteresis := rResetHysteresis;
    _bTreatSensorFaultAsTrip := bTreatSensorFaultAsTrip;

    _bInitialized := TRUE;
    _fbError.Clear();
    Init := TRUE;
END_METHOD

METHOD PUBLIC Execute: BOOL
    IF NOT _bInitialized THEN
        RETURN;
    END_IF

    // 1. Read the independent safety sensor (lifecycle owned by wiring program)
    _rTemperature := _ipSafetyTc.GetMeasurement();
    _bSensorFault := _ipSafetyTc.IsError();

    // 2. Over-temperature trip (latching)
    IF NOT _bTripLatched THEN
        IF _rTemperature > _rTripLimit THEN
            _bTripLatched := TRUE;
            _fbError.RaiseWithValues(
                E_ErrorId.ERR_CTRL_LIMIT_EXCEEDED,
                'SafetyTC',
                _rTemperature,
                _rTripLimit,
                'C');
        ELSIF _bSensorFault AND _bTreatSensorFaultAsTrip THEN
            // Fail-safe: loss of the safety sensor is itself a trip
            _bTripLatched := TRUE;
            _fbError.RaiseFromChild(_ipSafetyTc.GetError());
        END_IF
    END_IF

    // 3. Determine whether reset is permitted (cooled below limit - hysteresis, fault-free)
    _bCanReset := _bTripLatched
        AND NOT _bSensorFault
        AND (_rTemperature < (_rTripLimit - _rResetHysteresis));

    // 4. Update block reason (operator feedback)
    IF NOT _bTripLatched THEN
        _sBlockReason := '';
    ELSIF _bSensorFault THEN
        _sBlockReason := 'Safety TC fault';
    ELSIF _rTemperature >= (_rTripLimit - _rResetHysteresis) THEN
        _sBlockReason := 'Temperature still above reset threshold';
    ELSE
        _sBlockReason := '';
    END_IF

    Execute := NOT _bTripLatched;
END_METHOD

METHOD PUBLIC Reset: BOOL
    IF NOT _bTripLatched THEN
        Reset := TRUE; // Already clear
        RETURN;
    END_IF

    IF _bCanReset THEN
        _bTripLatched := FALSE;
        _sBlockReason := '';
        _fbError.Clear();
        Reset := TRUE;
    ELSE
        Reset := FALSE;
    END_IF
END_METHOD

METHOD PUBLIC IsTripActive: BOOL
    IsTripActive := _bTripLatched;
END_METHOD

METHOD PUBLIC CanReset: BOOL
    CanReset := _bCanReset;
END_METHOD

METHOD PUBLIC GetBlockReason: STRING(80)
    GetBlockReason := _sBlockReason;
END_METHOD

METHOD PUBLIC GetError: ST_Error
    GetError := _fbError.GetError();
END_METHOD

METHOD PUBLIC GetTemperature: LREAL
    GetTemperature := _rTemperature;
END_METHOD

METHOD PUBLIC IsInitialized: BOOL
    IsInitialized := _bInitialized;
END_METHOD

END_FUNCTION_BLOCK
